// TwinCAT 3 PLC project PLC1
// ProgramVersion: 3.1.4023.0
// libraries:
//   HomePLC Alarm Manager, * (Tom Oyen)
//   HomePLC DIO, * (Tom Oyen)
//   HomePLC Home, * (Tom Oyen)
//   HomePLC Logging, * (Tom Oyen)
//   Tc2_Standard, * (Beckhoff Automation GmbH)
//   Tc2_System, * (Beckhoff Automation GmbH)
//   Tc3_Module, * (Beckhoff Automation GmbH)
//   VisuDialogs, * (System)
//   HomePLC Link Manager,newest,Tom Oyen
// project tree:
//   / Class Diagram.TcCD (not stored), GlobalTextList.TcGTLO, PlcTask.TcTTO, Visualization Manager.TcVMO (not stored)
//   DUTs/Areas/ ST_Area_DiningRoom.TcDUT, ST_Area_Bedroom2.TcDUT, ST_Area_Toilet2.TcDUT, ST_Area_Bathroom.TcDUT, ST_Area_Bedroom1.TcDUT, ST_Area_Entrance.TcDUT, ST_Area_Kitchen.TcDUT, ST_Area_StorageRoom.TcDUT, ST_Area_Toilet1.TcDUT, ST_Area_LivingRoom.TcDUT
//   DUTs/Floors/ ST_Floor_FirstFloor.TcDUT, ST_Floor_SecondFloor.TcDUT
//   DUTs/Wall plates/ ST_WP_EntranceDoor.TcDUT, ST_WP_EntranceStairs.TcDUT, ST_WP_StorageRoom.TcDUT, ST_WP_Bathroom.TcDUT, ST_WP_Bedroom1.TcDUT, ST_WP_Bedroom1BedR.TcDUT, ST_WP_Bedroom1BedL.TcDUT, ST_WP_Bedroom2.TcDUT, ST_WP_Toilet2.TcDUT, ST_WP_LivingRoom.TcDUT, ST_WP_Toilet1.TcDUT, ST_WP_DiningRoom.TcDUT, ST_WP_Kitchen.TcDUT
//   GVLs/ IO.TcGVL
//   POUs/General/Implicit checks/ CheckBounds.TcPOU, CheckDivDInt.TcPOU, CheckDivLInt.TcPOU, CheckDivLReal.TcPOU, CheckDivReal.TcPOU, CheckLRangeSigned.TcPOU, CheckLRangeUnsigned.TcPOU, CheckPointer.TcPOU, CheckRangeSigned.TcPOU, CheckRangeUnsigned.TcPOU
//   POUs/Home/ FB_MyHome.TcPOU
//   POUs/ MAIN.TcPOU
//   POUs/Simulation/ FB_ButtonSim.TcPOU, FB_Simulation.TcPOU
//   VISUs/ Alarm.TcVIS, LinkInfo.TcVIS, Overview.TcVIS
// real-time tasks:
//   TASK PlcTask: cycle T#10ms, priority 20, ADS port 350
//   TASK VISU_TASK: cycle T#200000us, priority 30, ADS port 351

CONFIGURATION PLC1
    RESOURCE PLC ON TwinCAT3
        TASK PlcTask(INTERVAL := T#10ms, PRIORITY := 20);
        PROGRAM MAIN WITH PlcTask : MAIN;
    END_RESOURCE
END_CONFIGURATION

// ---- DUTs/Areas/ST_Area_DiningRoom.TcDUT
TYPE ST_Area_DiningRoom :
STRUCT
	wpRoom				: ST_WP_DiningRoom;
	fbSpotLights		: FB_DigitalOut;
	fbCenterLight		: FB_DigitalOut;
	fbAlarmsensor		: FB_AlarmSensor(sSensorName := 'DiningRoom', bEnableWarning := TRUE);
END_STRUCT
END_TYPE

// ---- DUTs/Areas/ST_Area_Bedroom2.TcDUT
TYPE ST_Area_Bedroom2 :
STRUCT
	wpRoom				: ST_WP_Bedroom2;
	fbSpotLights		: FB_DigitalOut;
END_STRUCT
END_TYPE

// ---- DUTs/Areas/ST_Area_Toilet2.TcDUT
TYPE ST_Area_Toilet2 :
STRUCT
	wpRuimte			: ST_WP_Toilet2;		// WC2 B1L0
	fbLichtSpot			: FB_DigitalOut;	// Licht spot + nis spot
END_STRUCT
END_TYPE

// ---- DUTs/Areas/ST_Area_Bathroom.TcDUT
TYPE ST_Area_Bathroom :
STRUCT
	wpRoom				: ST_WP_Bathroom;
	fbSpotLights		: FB_DigitalOut;
	fbSinkLights		: FB_DigitalOut;
END_STRUCT
END_TYPE

// ---- DUTs/Areas/ST_Area_Bedroom1.TcDUT
TYPE ST_Area_Bedroom1 :
STRUCT
	wpRoom				: ST_WP_Bedroom1;
	wpBedL				: ST_WP_Bedroom1BedL;
	fbSocketBedL		: FB_DigitalOut;
	wpBedR				: ST_WP_Bedroom1BedR;
	fbSocketBedR		: FB_DigitalOut;
	fbSpotLights		: FB_DigitalOut;
END_STRUCT
END_TYPE

// ---- DUTs/Floors/ST_Floor_FirstFloor.TcDUT
TYPE ST_Floor_FirstFloor :
STRUCT
	Entrance			: ST_Area_Entrance;
	Toilet1				: ST_Area_Toilet1;
	LivingRoom			: ST_Area_LivingRoom;
	DiningRoom			: ST_Area_DiningRoom;
	Kitchen				: ST_Area_Kitchen;
	StorageRoom			: ST_Area_StorageRoom;
END_STRUCT
END_TYPE

// ---- DUTs/Floors/ST_Floor_SecondFloor.TcDUT
TYPE ST_Floor_SecondFloor :
STRUCT
	Toilet2				: ST_Area_Toilet2;
	Bathroom			: ST_Area_Bathroom;
	Bedroom1			: ST_Area_Bedroom1;
	Bedroom2			: ST_Area_Bedroom2;
END_STRUCT
END_TYPE

// ---- DUTs/Areas/ST_Area_Entrance.TcDUT
TYPE ST_Area_Entrance :
STRUCT
	wpDoor				: ST_WP_EntranceDoor;
	fbAlarmPanel		: FB_AlarmKeypad(sKeypadName := 'Entrance');
	wpStairs			: ST_WP_EntranceStairs;
	fbSpotLights		: FB_DigitalOut;
	fbAlarmSensor		: FB_AlarmSensor(sSensorName := 'Entrance', bEnableWarning := TRUE);
	fbAlarmSiren		: FB_AlarmSiren(sSirenName := 'Entrance');
END_STRUCT
END_TYPE

// ---- DUTs/Areas/ST_Area_Kitchen.TcDUT
TYPE ST_Area_Kitchen :
STRUCT
	wpRoom				: ST_WP_Kitchen;
	fbLightIsland		: FB_DigitalOut;
	fbCenterLight		: FB_DigitalOut;
	fbSocket			: FB_DigitalOut;
	fbAlarmSensor		: FB_AlarmSensor(sSensorName := 'Kitchen', bEnableWarning := TRUE);
END_STRUCT
END_TYPE

// ---- DUTs/Areas/ST_Area_StorageRoom.TcDUT
TYPE ST_Area_StorageRoom :
STRUCT
	wpRoom				: ST_WP_StorageRoom;
	fbSpotLights		: FB_DigitalOut;
	fbAlarmsensor		: FB_AlarmSensor(sSensorName := 'StorageRoom', bEnableWarning := FALSE);
END_STRUCT
END_TYPE

// ---- DUTs/Areas/ST_Area_Toilet1.TcDUT
TYPE ST_Area_Toilet1 :
STRUCT
	wpRoom				: ST_WP_Toilet1;
	fbSpotLight			: FB_DigitalOut;
END_STRUCT
END_TYPE

// ---- DUTs/Areas/ST_Area_LivingRoom.TcDUT
TYPE ST_Area_LivingRoom :
STRUCT
	wpRoom			: ST_WP_LivingRoom;
	fbSpotLights	: FB_DigitalOut;
	fbAlarmSensor	: FB_AlarmSensor(sSensorName := 'LivingRoom', bEnableWarning := FALSE);
END_STRUCT
END_TYPE

// ---- DUTs/Wall plates/ST_WP_EntranceDoor.TcDUT
// Inkom deur - B11-11L11-11
TYPE ST_WP_EntranceDoor :
STRUCT
	fbButton1		: FB_DigitalIn;
	fbLed1			: FB_DigitalOut;
	fbButton2		: FB_DigitalIn;
	fbLed2			: FB_DigitalOut;
	fbButton3		: FB_DigitalIn;
	fbLed3			: FB_DigitalOut;
	fbButton4		: FB_DigitalIn;
	fbLed4			: FB_DigitalOut;
END_STRUCT
END_TYPE

// ---- DUTs/Wall plates/ST_WP_EntranceStairs.TcDUT
// Inkom trap B1-11L0-00
TYPE ST_WP_EntranceStairs :
STRUCT
	fbButton1		: FB_DigitalIn;
	fbButton2		: FB_DigitalIn;
	fbButton3		: FB_DigitalIn;
END_STRUCT
END_TYPE

// ---- DUTs/Wall plates/ST_WP_StorageRoom.TcDUT
// Bergplaats B1-11L0-00
TYPE ST_WP_StorageRoom :
STRUCT
	fbButton1		: FB_DigitalIn;
	fbButton2		: FB_DigitalIn;
	fbButton3		: FB_DigitalIn;
END_STRUCT
END_TYPE

// ---- DUTs/Wall plates/ST_WP_Bathroom.TcDUT
// Badkamer meubel B1L0
TYPE ST_WP_Bathroom :
STRUCT
	fbKnop1		: FB_DigitalIn;
END_STRUCT
END_TYPE

// ---- DUTs/Wall plates/ST_WP_Bedroom1.TcDUT
// Slaapkamer 1 B1-1L0-0
TYPE ST_WP_Bedroom1 :
STRUCT
	fbButton1		: FB_DigitalIn;
	fbButton2		: FB_DigitalIn;
END_STRUCT
END_TYPE

// ---- DUTs/Wall plates/ST_WP_Bedroom1BedR.TcDUT
// Slaapkamer 1 bed R B11L00
TYPE ST_WP_Bedroom1BedR :
STRUCT
	fbButton1		: FB_DigitalIn;
	fbButton2		: FB_DigitalIn;
END_STRUCT
END_TYPE

// ---- DUTs/Wall plates/ST_WP_Bedroom1BedL.TcDUT
// Slaapkamer 1 bed L B11L00
TYPE ST_WP_Bedroom1BedL :
STRUCT
	fbButton1		: FB_DigitalIn;
	fbButton2		: FB_DigitalIn;
END_STRUCT
END_TYPE

// ---- DUTs/Wall plates/ST_WP_Bedroom2.TcDUT
// Slaapkamer 2 B1L0
TYPE ST_WP_Bedroom2 :
STRUCT
	fbButton1		: FB_DigitalIn;
END_STRUCT
END_TYPE

// ---- DUTs/Wall plates/ST_WP_Toilet2.TcDUT
// WC2 B1L0
TYPE ST_WP_Toilet2 :
STRUCT
	fbButton1		: FB_DigitalIn;
END_STRUCT
END_TYPE

// ---- DUTs/Wall plates/ST_WP_LivingRoom.TcDUT
// Zithoek B11-11L00-00
TYPE ST_WP_LivingRoom :
STRUCT
	fbButton1		: FB_DigitalIn;
	fbButton2		: FB_DigitalIn;
	fbButton3		: FB_DigitalIn;
	fbButton4		: FB_DigitalIn;
END_STRUCT
END_TYPE

// ---- DUTs/Wall plates/ST_WP_Toilet1.TcDUT
// WC1 B1L0
TYPE ST_WP_Toilet1 :
STRUCT
	fbButton1		: FB_DigitalIn;
END_STRUCT
END_TYPE

// ---- DUTs/Wall plates/ST_WP_DiningRoom.TcDUT
// Eethoek B1-1-11L0-0-00
TYPE ST_WP_DiningRoom :
STRUCT
	fbKnop1		: FB_DigitalIn;
	fbKnop2		: FB_DigitalIn;
	fbKnop3		: FB_DigitalIn;
	fbKnop4		: FB_DigitalIn;
END_STRUCT
END_TYPE

// ---- DUTs/Wall plates/ST_WP_Kitchen.TcDUT
// Keuken B1-11-11L0-00-00
TYPE ST_WP_Kitchen :
STRUCT
	fbButton1		: FB_DigitalIn;
	fbButton2		: FB_DigitalIn;
	fbButton3		: FB_DigitalIn;
	fbButton4		: FB_DigitalIn;
	fbButton5		: FB_DigitalIn;
END_STRUCT
END_TYPE

// ---- GVLs/IO.TcGVL
{attribute 'qualified_only'}
VAR_GLOBAL
	// IO
	FirstFloor		: ST_Floor_FirstFloor;
	SecondFloor		: ST_Floor_SecondFloor;
END_VAR

// ---- POUs/MAIN.TcPOU
// Home PLC
PROGRAM MAIN
VAR
	fbHome			: FB_MyHome;
	fbSimulation	: FB_Simulation;
END_VAR

fbHome.Execute();
//fbSimulation.Execute();

END_PROGRAM

// ---- POUs/Home/FB_MyHome.TcPOU
// Home implementation
FUNCTION_BLOCK FB_MyHome EXTENDS FB_Home
VAR
	// IO groups
	fbDIGroupAllOff		: FB_DIGroup;		// Input group containing all inputs for the all-off function
	fbDOGroupAllOff		: FB_DOGroup;		// Output group containing all outputs for the all-off function
END_VAR

// Configure
METHOD PROTECTED Configure
CreateDIGroupAllOff(IDIGroup := fbDIGroupAllOff);
CreateDOGroupAllOff(IDOGroup := fbDOGroupAllOff);

SUPER^.Configure();
END_METHOD

// Configure alarm
METHOD PROTECTED ConfigureAlarm
VAR_INPUT
	IAlarmManager	: I_AlarmManager;		// Alarm manager interface
END_VAR
IAlarmManager.AddKeypad(IKeyPad := IO.FirstFloor.Entrance.fbAlarmPanel);

IAlarmManager.AddSensor(ISensor := IO.FirstFloor.Entrance.fbAlarmSensor);
IAlarmManager.AddSensor(ISensor := IO.FirstFloor.LivingRoom.fbAlarmSensor);
IAlarmManager.AddSensor(ISensor := IO.FirstFloor.DiningRoom.fbAlarmsensor);
IAlarmManager.AddSensor(ISensor := IO.FirstFloor.Kitchen.fbAlarmSensor);
IAlarmManager.AddSensor(ISensor := IO.FirstFloor.StorageRoom.fbAlarmsensor);

IAlarmManager.AddSiren(ISiren := IO.FirstFloor.Entrance.fbAlarmSiren);
END_METHOD

// Add links
METHOD PROTECTED ConfigureLinks
VAR_INPUT
	ILinkManager	: I_LinkManager;		// Link manager interface
END_VAR
// All off
ILinkManager.Link.InputGroup := fbDIGroupAllOff;
ILinkManager.Link.OutputGroup := fbDOGroupAllOff;
ILinkManager.Link.OutputReaction.OnHold := E_DOCommand.Off;
ILinkManager.Link.ExcludeFromOverview := TRUE;
ILinkManager.CommitLink();

// First floor - entrance spot lights
ILinkManager.Link.InputGroup.AddInput(IO.FirstFloor.Entrance.wpDoor.fbButton4);
ILinkManager.Link.InputGroup.AddInput(IO.FirstFloor.Entrance.wpStairs.fbButton3);
ILinkManager.Link.InputGroup.AddInput(IO.FirstFloor.StorageRoom.wpRoom.fbButton1);
ILinkManager.Link.OutputReaction.OnShortPress := E_DOCommand.Toggle;
ILinkManager.Link.OutputGroup.AddOutput(IO.FirstFloor.Entrance.fbSpotLights);
ILinkManager.Link.OutputGroup.AddIndicator(IO.FirstFloor.Entrance.wpDoor.fbLed4);
ILinkManager.CommitLink();

// First floor - WC1 spot light
ILinkManager.Link.InputGroup.AddInput(IO.FirstFloor.Toilet1.wpRoom.fbButton1);
ILinkManager.Link.OutputReaction.OnShortPress := E_DOCommand.Toggle;
ILinkManager.Link.OutputGroup.AddOutput(IO.FirstFloor.Toilet1.fbSpotLight);
ILinkManager.CommitLink();

// First floor - Living room spot lights
ILinkManager.Link.InputGroup.AddInput(IO.FirstFloor.LivingRoom.wpRoom.fbButton4);
ILinkManager.Link.InputGroup.AddInput(IO.FirstFloor.DiningRoom.wpRoom.fbKnop4);
ILinkManager.Link.InputGroup.AddInput(IO.FirstFloor.Entrance.wpStairs.fbButton2);
ILinkManager.Link.OutputReaction.OnShortPress := E_DOCommand.Toggle;
ILinkManager.Link.OutputGroup.AddOutput(IO.FirstFloor.LivingRoom.fbSpotLights);
ILinkManager.CommitLink();

// First floor - Dining room spot lights
ILinkManager.Link.InputGroup.AddInput(IO.FirstFloor.DiningRoom.wpRoom.fbKnop3);
ILinkManager.Link.InputGroup.AddInput(IO.FirstFloor.LivingRoom.wpRoom.fbButton1);
ILinkManager.Link.OutputReaction.OnShortPress := E_DOCommand.Toggle;
ILinkManager.Link.OutputGroup.AddOutput(IO.FirstFloor.DiningRoom.fbSpotLights);
ILinkManager.CommitLink();

// First floor - Dining room center light
ILinkManager.Link.InputGroup.AddInput(IO.FirstFloor.DiningRoom.wpRoom.fbKnop2);
ILinkManager.Link.InputGroup.AddInput(IO.FirstFloor.LivingRoom.wpRoom.fbButton2);
ILinkManager.Link.OutputReaction.OnShortPress := E_DOCommand.Toggle;
ILinkManager.Link.OutputGroup.AddOutput(IO.FirstFloor.DiningRoom.fbCenterLight);
ILinkManager.CommitLink();

// First floor - Kitchen island lights
ILinkManager.Link.InputGroup.AddInput(IO.FirstFloor.Kitchen.wpRoom.fbButton4);
ILinkManager.Link.OutputReaction.OnShortPress := E_DOCommand.Toggle;
ILinkManager.Link.OutputGroup.AddOutput(IO.FirstFloor.Kitchen.fbLightIsland);
ILinkManager.CommitLink();

// First floor - Kitchen center light
ILinkManager.Link.InputGroup.AddInput(IO.FirstFloor.Kitchen.wpRoom.fbButton2);
ILinkManager.Link.OutputReaction.OnShortPress := E_DOCommand.Toggle;
ILinkManager.Link.OutputGroup.AddOutput(IO.FirstFloor.Kitchen.fbCenterLight);
ILinkManager.CommitLink();

// First floor - Kitchen socket
ILinkManager.Link.InputGroup.AddInput(IO.FirstFloor.Kitchen.wpRoom.fbButton5);
ILinkManager.Link.OutputReaction.OnShortPress := E_DOCommand.Toggle;
ILinkManager.Link.OutputGroup.AddOutput(IO.FirstFloor.Kitchen.fbSocket);
ILinkManager.CommitLink();

// First floor - Storage room spot lights
ILinkManager.Link.InputGroup.AddInput(IO.FirstFloor.StorageRoom.wpRoom.fbButton2);
ILinkManager.Link.OutputReaction.OnShortPress := E_DOCommand.Toggle;
ILinkManager.Link.OutputGroup.AddOutput(IO.FirstFloor.StorageRoom.fbSpotLights);
ILinkManager.CommitLink();

// Second floor - WC2 spots
ILinkManager.Link.InputGroup.AddInput(IO.SecondFloor.Toilet2.wpRuimte.fbButton1);
ILinkManager.Link.OutputReaction.OnShortPress := E_DOCommand.Toggle;
ILinkManager.Link.OutputGroup.AddOutput(IO.SecondFloor.Toilet2.fbLichtSpot);
ILinkManager.CommitLink();

// Second floor - Bathroom sink lights
ILinkManager.Link.InputGroup.AddInput(IO.SecondFloor.Bathroom.wpRoom.fbKnop1);
ILinkManager.Link.OutputReaction.OnShortPress := E_DOCommand.Toggle;
ILinkManager.Link.OutputGroup.AddOutput(IO.SecondFloor.Bathroom.fbSinkLights);
ILinkManager.CommitLink();

// Second floor - Bedroom 1 spot lights
ILinkManager.Link.InputGroup.AddInput(IO.SecondFloor.Bedroom1.wpRoom.fbButton2);
ILinkManager.Link.InputGroup.AddInput(IO.SecondFloor.Bedroom1.wpBedL.fbButton1);
ILinkManager.Link.InputGroup.AddInput(IO.SecondFloor.Bedroom1.wpBedR.fbButton2);
ILinkManager.Link.OutputReaction.OnShortPress := E_DOCommand.Toggle;
ILinkManager.Link.OutputGroup.AddOutput(IO.SecondFloor.Bedroom1.fbSpotLights);
ILinkManager.CommitLink();

// Second floor - Bedroom 1 socket L
ILinkManager.Link.InputGroup.AddInput(IO.SecondFloor.Bedroom1.wpBedL.fbButton2);
ILinkManager.Link.OutputReaction.OnShortPress := E_DOCommand.Toggle;
ILinkManager.Link.OutputGroup.AddOutput(IO.SecondFloor.Bedroom1.fbSocketBedL);
ILinkManager.CommitLink();

// Second floor - Bedroom 1 socket R
ILinkManager.Link.InputGroup.AddInput(IO.SecondFloor.Bedroom1.wpBedR.fbButton1);
ILinkManager.Link.OutputReaction.OnShortPress := E_DOCommand.Toggle;
ILinkManager.Link.OutputGroup.AddOutput(IO.SecondFloor.Bedroom1.fbSocketBedR);
ILinkManager.CommitLink();

// Second floor - Bedroom 2 spots
ILinkManager.Link.InputGroup.AddInput(IO.SecondFloor.Bedroom2.wpRoom.fbButton1);
ILinkManager.Link.OutputReaction.OnShortPress := E_DOCommand.Toggle;
ILinkManager.Link.OutputGroup.AddOutput(IO.SecondFloor.Bedroom2.fbSpotLights);
ILinkManager.CommitLink();
END_METHOD

// Create DI group of all inputs (used to call all Execute methods)
METHOD PROTECTED CreateDIGroupAll
VAR_INPUT
	IDIGroup	: I_DIGroup;		// Digital input group interface
END_VAR
// First floor
IDIGroup.AddInput(IO.FirstFloor.StorageRoom.wpRoom.fbButton1);
IDIGroup.AddInput(IO.FirstFloor.StorageRoom.wpRoom.fbButton2);
IDIGroup.AddInput(IO.FirstFloor.StorageRoom.wpRoom.fbButton3);
IDIGroup.AddInput(IO.FirstFloor.DiningRoom.wpRoom.fbKnop1);
IDIGroup.AddInput(IO.FirstFloor.DiningRoom.wpRoom.fbKnop2);
IDIGroup.AddInput(IO.FirstFloor.DiningRoom.wpRoom.fbKnop3);
IDIGroup.AddInput(IO.FirstFloor.DiningRoom.wpRoom.fbKnop4);
IDIGroup.AddInput(IO.FirstFloor.Entrance.wpDoor.fbButton1);
IDIGroup.AddInput(IO.FirstFloor.Entrance.wpDoor.fbButton2);
IDIGroup.AddInput(IO.FirstFloor.Entrance.wpDoor.fbButton3);
IDIGroup.AddInput(IO.FirstFloor.Entrance.wpDoor.fbButton4);
IDIGroup.AddInput(IO.FirstFloor.Entrance.wpStairs.fbButton1);
IDIGroup.AddInput(IO.FirstFloor.Entrance.wpStairs.fbButton2);
IDIGroup.AddInput(IO.FirstFloor.Entrance.wpStairs.fbButton3);
IDIGroup.AddInput(IO.FirstFloor.Kitchen.wpRoom.fbButton1);
IDIGroup.AddInput(IO.FirstFloor.Kitchen.wpRoom.fbButton2);
IDIGroup.AddInput(IO.FirstFloor.Kitchen.wpRoom.fbButton3);
IDIGroup.AddInput(IO.FirstFloor.Kitchen.wpRoom.fbButton4);
IDIGroup.AddInput(IO.FirstFloor.Kitchen.wpRoom.fbButton5);
IDIGroup.AddInput(IO.FirstFloor.Toilet1.wpRoom.fbButton1);
IDIGroup.AddInput(IO.FirstFloor.LivingRoom.wpRoom.fbButton1);
IDIGroup.AddInput(IO.FirstFloor.LivingRoom.wpRoom.fbButton2);
IDIGroup.AddInput(IO.FirstFloor.LivingRoom.wpRoom.fbButton3);
IDIGroup.AddInput(IO.FirstFloor.LivingRoom.wpRoom.fbButton4);

// Verdieping
IDIGroup.AddInput(IO.SecondFloor.Bathroom.wpRoom.fbKnop1);
IDIGroup.AddInput(IO.SecondFloor.Bedroom1.wpBedL.fbButton1);
IDIGroup.AddInput(IO.SecondFloor.Bedroom1.wpBedL.fbButton2);
IDIGroup.AddInput(IO.SecondFloor.Bedroom1.wpBedR.fbButton1);
IDIGroup.AddInput(IO.SecondFloor.Bedroom1.wpBedR.fbButton2);
IDIGroup.AddInput(IO.SecondFloor.Bedroom1.wpRoom.fbButton1);
IDIGroup.AddInput(IO.SecondFloor.Bedroom1.wpRoom.fbButton2);
IDIGroup.AddInput(IO.SecondFloor.Bedroom2.wpRoom.fbButton1);
IDIGroup.AddInput(IO.SecondFloor.Toilet2.wpRuimte.fbButton1);


// Alarm
// Included here so these buttons can be used for general commands as well (e.g. all off)
IDIGroup.AddInput(IO.FirstFloor.Entrance.fbAlarmPanel.fbButton1);
IDIGroup.AddInput(IO.FirstFloor.Entrance.fbAlarmPanel.fbButton2);
IDIGroup.AddInput(IO.FirstFloor.Entrance.fbAlarmPanel.fbButton3);
IDIGroup.AddInput(IO.FirstFloor.Entrance.fbAlarmPanel.fbButton4);
IDIGroup.AddInput(IO.FirstFloor.Entrance.fbAlarmPanel.fbButton5);
IDIGroup.AddInput(IO.FirstFloor.Entrance.fbAlarmPanel.fbButton6);
END_METHOD

// Create DI group of all inputs that are used to turn all outputs off
METHOD PRIVATE CreateDIGroupAllOff
VAR_INPUT
	IDIGroup	: I_DIGroup;		// Digital input group interface
END_VAR
// Gelijkvloers
IDIGroup.AddInput(IO.FirstFloor.StorageRoom.wpRoom.fbButton1);
IDIGroup.AddInput(IO.FirstFloor.StorageRoom.wpRoom.fbButton2);
IDIGroup.AddInput(IO.FirstFloor.StorageRoom.wpRoom.fbButton3);
IDIGroup.AddInput(IO.FirstFloor.DiningRoom.wpRoom.fbKnop1);
IDIGroup.AddInput(IO.FirstFloor.DiningRoom.wpRoom.fbKnop2);
IDIGroup.AddInput(IO.FirstFloor.DiningRoom.wpRoom.fbKnop3);
IDIGroup.AddInput(IO.FirstFloor.DiningRoom.wpRoom.fbKnop4);
IDIGroup.AddInput(IO.FirstFloor.Entrance.wpDoor.fbButton1);
IDIGroup.AddInput(IO.FirstFloor.Entrance.wpDoor.fbButton2);
IDIGroup.AddInput(IO.FirstFloor.Entrance.wpDoor.fbButton3);
IDIGroup.AddInput(IO.FirstFloor.Entrance.wpDoor.fbButton4);
IDIGroup.AddInput(IO.FirstFloor.Entrance.wpStairs.fbButton1);
IDIGroup.AddInput(IO.FirstFloor.Entrance.wpStairs.fbButton2);
IDIGroup.AddInput(IO.FirstFloor.Entrance.wpStairs.fbButton3);
IDIGroup.AddInput(IO.FirstFloor.Kitchen.wpRoom.fbButton1);
IDIGroup.AddInput(IO.FirstFloor.Kitchen.wpRoom.fbButton2);
IDIGroup.AddInput(IO.FirstFloor.Kitchen.wpRoom.fbButton3);
IDIGroup.AddInput(IO.FirstFloor.Kitchen.wpRoom.fbButton4);
IDIGroup.AddInput(IO.FirstFloor.Kitchen.wpRoom.fbButton5);
IDIGroup.AddInput(IO.FirstFloor.Toilet1.wpRoom.fbButton1);
IDIGroup.AddInput(IO.FirstFloor.LivingRoom.wpRoom.fbButton1);
IDIGroup.AddInput(IO.FirstFloor.LivingRoom.wpRoom.fbButton2);
IDIGroup.AddInput(IO.FirstFloor.LivingRoom.wpRoom.fbButton3);
IDIGroup.AddInput(IO.FirstFloor.LivingRoom.wpRoom.fbButton4);

// Verdieping
IDIGroup.AddInput(IO.SecondFloor.Bathroom.wpRoom.fbKnop1);
IDIGroup.AddInput(IO.SecondFloor.Bedroom1.wpBedL.fbButton1);
IDIGroup.AddInput(IO.SecondFloor.Bedroom1.wpBedL.fbButton2);
IDIGroup.AddInput(IO.SecondFloor.Bedroom1.wpBedR.fbButton1);
IDIGroup.AddInput(IO.SecondFloor.Bedroom1.wpBedR.fbButton2);
IDIGroup.AddInput(IO.SecondFloor.Bedroom1.wpRoom.fbButton1);
IDIGroup.AddInput(IO.SecondFloor.Bedroom1.wpRoom.fbButton2);
IDIGroup.AddInput(IO.SecondFloor.Bedroom2.wpRoom.fbButton1);
IDIGroup.AddInput(IO.SecondFloor.Toilet2.wpRuimte.fbButton1);

// Alarm
IDIGroup.AddInput(IO.FirstFloor.Entrance.fbAlarmPanel.fbButton1);
IDIGroup.AddInput(IO.FirstFloor.Entrance.fbAlarmPanel.fbButton2);
IDIGroup.AddInput(IO.FirstFloor.Entrance.fbAlarmPanel.fbButton3);
IDIGroup.AddInput(IO.FirstFloor.Entrance.fbAlarmPanel.fbButton4);
IDIGroup.AddInput(IO.FirstFloor.Entrance.fbAlarmPanel.fbButton5);
IDIGroup.AddInput(IO.FirstFloor.Entrance.fbAlarmPanel.fbButton6);
END_METHOD

// Create DO group of all outputs (used to call all Execute methods)
METHOD PROTECTED CreateDOGroupAll
VAR_INPUT
	IDOGroup	: I_DOGroup;		// Digital output group interface
END_VAR
// First floor
IDOGroup.AddOutput(IO.FirstFloor.StorageRoom.fbSpotLights);
IDOGroup.AddOutput(IO.FirstFloor.DiningRoom.fbSpotLights);
IDOGroup.AddOutput(IO.FirstFloor.DiningRoom.fbCenterLight);
IDOGroup.AddOutput(IO.FirstFloor.Entrance.fbSpotLights);
IDOGroup.AddOutput(IO.FirstFloor.Entrance.wpDoor.fbLed1);
IDOGroup.AddOutput(IO.FirstFloor.Entrance.wpDoor.fbLed2);
IDOGroup.AddOutput(IO.FirstFloor.Entrance.wpDoor.fbLed3);
IDOGroup.AddOutput(IO.FirstFloor.Entrance.wpDoor.fbLed4);
IDOGroup.AddOutput(IO.FirstFloor.Kitchen.fbLightIsland);
IDOGroup.AddOutput(IO.FirstFloor.Kitchen.fbCenterLight);
IDOGroup.AddOutput(IO.FirstFloor.Kitchen.fbSocket);
IDOGroup.AddOutput(IO.FirstFloor.Toilet1.fbSpotLight);
IDOGroup.AddOutput(IO.FirstFloor.LivingRoom.fbSpotLights);

// Second floor
IDOGroup.AddOutput(IO.SecondFloor.Bathroom.fbSpotLights);
IDOGroup.AddOutput(IO.SecondFloor.Bathroom.fbSinkLights);
IDOGroup.AddOutput(IO.SecondFloor.Bedroom1.fbSpotLights);
IDOGroup.AddOutput(IO.SecondFloor.Bedroom1.fbSocketBedL);
IDOGroup.AddOutput(IO.SecondFloor.Bedroom1.fbSocketBedR);
IDOGroup.AddOutput(IO.SecondFloor.Bedroom2.fbSpotLights);
IDOGroup.AddOutput(IO.SecondFloor.Toilet2.fbLichtSpot);


// Alarm
IDOGroup.AddOutput(IO.FirstFloor.Entrance.fbAlarmPanel.fbLed1);
IDOGroup.AddOutput(IO.FirstFloor.Entrance.fbAlarmPanel.fbLed2);
IDOGroup.AddOutput(IO.FirstFloor.Entrance.fbAlarmPanel.fbLed3);
IDOGroup.AddOutput(IO.FirstFloor.Entrance.fbAlarmPanel.fbLed4);
IDOGroup.AddOutput(IO.FirstFloor.Entrance.fbAlarmPanel.fbLed5);
IDOGroup.AddOutput(IO.FirstFloor.Entrance.fbAlarmPanel.fbLed6);
IDOGroup.AddOutput(IO.FirstFloor.Entrance.fbAlarmPanel.fbBuzzer);
IDOGroup.AddOutput(IO.FirstFloor.Entrance.fbAlarmSiren.fbSiren);
IDOGroup.AddOutput(IO.FirstFloor.Entrance.fbAlarmSiren.fbLight);
END_METHOD

// Create DO group of all outputs that are turned off when all needs to be turned off
METHOD PRIVATE CreateDOGroupAllOff
VAR_INPUT
	IDOGroup	: I_DOGroup;		// Digital output group interface
END_VAR
// First floor
IDOGroup.AddOutput(IO.FirstFloor.StorageRoom.fbSpotLights);
IDOGroup.AddOutput(IO.FirstFloor.DiningRoom.fbSpotLights);
IDOGroup.AddOutput(IO.FirstFloor.DiningRoom.fbCenterLight);
IDOGroup.AddOutput(IO.FirstFloor.Entrance.fbSpotLights);
IDOGroup.AddOutput(IO.FirstFloor.Entrance.wpDoor.fbLed1);
IDOGroup.AddOutput(IO.FirstFloor.Entrance.wpDoor.fbLed2);
IDOGroup.AddOutput(IO.FirstFloor.Entrance.wpDoor.fbLed3);
IDOGroup.AddOutput(IO.FirstFloor.Entrance.wpDoor.fbLed4);
IDOGroup.AddOutput(IO.FirstFloor.Kitchen.fbLightIsland);
IDOGroup.AddOutput(IO.FirstFloor.Kitchen.fbCenterLight);
IDOGroup.AddOutput(IO.FirstFloor.Kitchen.fbSocket);
IDOGroup.AddOutput(IO.FirstFloor.Toilet1.fbSpotLight);
IDOGroup.AddOutput(IO.FirstFloor.LivingRoom.fbSpotLights);

// Verdieping
IDOGroup.AddOutput(IO.SecondFloor.Bathroom.fbSpotLights);
IDOGroup.AddOutput(IO.SecondFloor.Bathroom.fbSinkLights);
IDOGroup.AddOutput(IO.SecondFloor.Bedroom1.fbSpotLights);
IDOGroup.AddOutput(IO.SecondFloor.Bedroom1.fbSocketBedL);
IDOGroup.AddOutput(IO.SecondFloor.Bedroom1.fbSocketBedR);
IDOGroup.AddOutput(IO.SecondFloor.Bedroom2.fbSpotLights);
IDOGroup.AddOutput(IO.SecondFloor.Toilet2.fbLichtSpot);

// Alarm
IDOGroup.AddOutput(IO.FirstFloor.Entrance.fbAlarmPanel.fbBuzzer);
END_METHOD

END_FUNCTION_BLOCK

// ---- POUs/Simulation/FB_Simulation.TcPOU
FUNCTION_BLOCK FB_Simulation

METHOD Execute : BOOL
VAR_INST
	fbButton1		: FB_ButtonSim;
	fbButton2		: FB_ButtonSim;

	bShortPress1	: BOOL;
	bLongPress1		: BOOL;
	bHold1			: BOOL;
	
	bShortPress2	: BOOL;
	bLongPress2		: BOOL;
	bHold2			: BOOL;
END_VAR
fbButton1(IButton := IO.FirstFloor.Kitchen.wpRoom.fbButton1, bShortPress := bShortPress1, bLongPress := bLongPress1, bHold := bHold1);
fbButton2(IButton := IO.FirstFloor.Kitchen.wpRoom.fbButton2, bShortPress := bShortPress2, bLongPress := bLongPress2, bHold := bHold2);
END_METHOD

END_FUNCTION_BLOCK

// ---- POUs/Simulation/FB_ButtonSim.TcPOU
FUNCTION_BLOCK FB_ButtonSim
VAR_INPUT
	IButton			: I_DigitalIn;
END_VAR
VAR_IN_OUT
	bShortPress		: BOOL;
	bLongPress		: BOOL;
	bHold			: BOOL;
END_VAR
VAR
	bOut			: BOOL;
	fbTimer			: TON;
END_VAR

IF bShortPress	THEN fbTimer.PT := T#100MS; END_IF
IF bLongPress	THEN fbTimer.PT := T#500MS; END_IF
IF bHold		THEN fbTimer.PT := T#3000MS; END_IF
IF bShortPress OR bLongPress OR bHold THEN
	bOut := TRUE;
	bShortPress := FALSE;
	bLongPress := FALSE;
	bHold := FALSE;
END_IF

fbTimer(IN := bOut);
if fbTimer.Q then
	bOut := FALSE;
END_IF

IButton.SetExternalIn(bIn := bOut);

END_FUNCTION_BLOCK

// ---- POUs/General/Implicit checks/CheckBounds.TcPOU
// Implicitly generated code : DO NOT EDIT
FUNCTION CheckBounds : DINT
VAR_INPUT
	index, lower, upper: DINT;
END_VAR
// User defined local variables
VAR
    sMessageLow   : STRING := 'CheckBounds: Index too low (%d)';
    sMessageHigh  : STRING := 'CheckBounds: Index too high (%d)';
END_VAR

// This function is called every time an array is indexed
// See https://infosys.beckhoff.com/english.php?content=../content/1033/tc3_plc_intro/2530356875.html&id=

{noflow}
// Index too low
IF index < lower THEN
    CheckBounds := lower;
    // Log message
    ADSLOGDINT(msgCtrlMask := ADSLOG_MSGTYPE_WARN,
               msgFmtStr   := sMessageLow,
               dintArg     := index);

// Index too high
ELSIF index > upper THEN
    CheckBounds := upper;
    // Log message
    ADSLOGDINT(msgCtrlMask := ADSLOG_MSGTYPE_WARN,
               msgFmtStr   := sMessageHigh,
               dintArg     := index);

// Index OK
ELSE 
    CheckBounds := index;
END_IF
{flow}

END_FUNCTION

// ---- POUs/General/Implicit checks/CheckDivDInt.TcPOU
// Implicitly generated code : DO NOT EDIT
FUNCTION CheckDivDInt : DINT
VAR_INPUT
	divisor:DINT;
END_VAR
VAR
    sMessage   : STRING := 'CheckDivDInt: Division by zero (%d)';
END_VAR

// Implicitly generated code : Only an Implementation suggestion
{noflow}
IF divisor = 0 THEN
	CheckDivDInt:=1;
	// Log message
    ADSLOGDINT(msgCtrlMask := ADSLOG_MSGTYPE_WARN,
               msgFmtStr   := sMessage,
               dintArg     := divisor);
ELSE
	CheckDivDInt:=divisor;
END_IF;
{flow}

END_FUNCTION

// ---- POUs/General/Implicit checks/CheckDivLInt.TcPOU
// Implicitly generated code : DO NOT EDIT
FUNCTION CheckDivLInt : LINT
VAR_INPUT
	divisor:LINT;
END_VAR
VAR
    sMessage   : STRING := 'CheckDivLInt: Division by zero (%d)';
END_VAR

// Implicitly generated code : Only an Implementation suggestion
{noflow}
IF divisor = 0 THEN
	CheckDivLInt:=1;
	// Log message
    ADSLOGDINT(msgCtrlMask := ADSLOG_MSGTYPE_WARN,
               msgFmtStr   := sMessage,
               dintArg     := 0);
ELSE
	CheckDivLInt:=divisor;
END_IF;
{flow}

END_FUNCTION

// ---- POUs/General/Implicit checks/CheckDivLReal.TcPOU
// Implicitly generated code : DO NOT EDIT
FUNCTION CheckDivLReal : LREAL
VAR_INPUT
	divisor:LREAL;
END_VAR
VAR
    sMessage   : STRING := 'CheckDivLReal: Division by zero (%d)';
END_VAR

// Implicitly generated code : Only an Implementation suggestion
{noflow}
IF divisor = 0 THEN
	CheckDivLReal:=1;
	// Log message
    ADSLOGDINT(msgCtrlMask := ADSLOG_MSGTYPE_WARN,
               msgFmtStr   := sMessage,
               dintArg     := 0);
ELSE
	CheckDivLReal:=divisor;
END_IF;
{flow}

END_FUNCTION

// ---- POUs/General/Implicit checks/CheckDivReal.TcPOU
// Implicitly generated code : DO NOT EDIT
FUNCTION CheckDivReal : REAL
VAR_INPUT
	divisor:REAL;
END_VAR
VAR
    sMessage   : STRING := 'CheckDivReal: Division by zero (%d)';
END_VAR

// Implicitly generated code : Only an Implementation suggestion
{noflow}
IF divisor = 0 THEN
	CheckDivReal:=1;
	// Log message
    ADSLOGDINT(msgCtrlMask := ADSLOG_MSGTYPE_WARN,
               msgFmtStr   := sMessage,
               dintArg     := 0);
ELSE
	CheckDivReal:=divisor;
END_IF;
{flow}

END_FUNCTION

// ---- POUs/General/Implicit checks/CheckLRangeSigned.TcPOU
// Implicitly generated code : DO NOT EDIT
FUNCTION CheckLRangeSigned : LINT
VAR_INPUT
	value, lower, upper: LINT;
END_VAR
VAR
    sMessageLow   : STRING := 'CheckLRangeSigned: Value too low (%d)';
    sMessageHigh  : STRING := 'CheckLRangeSigned: Value too high (%d)';
END_VAR

// Implicitly generated code : Only an Implementation suggestion
{noflow}
IF (value < lower) THEN
	CheckLRangeSigned := lower;
	// Log message
    ADSLOGLREAL(msgCtrlMask := ADSLOG_MSGTYPE_WARN,
               msgFmtStr   := sMessageLow,
               lrealArg     := TO_REAL(value));
ELSIF(value > upper) THEN
	CheckLRangeSigned := upper;
	// Log message
    ADSLOGLREAL(msgCtrlMask := ADSLOG_MSGTYPE_WARN,
               msgFmtStr   := sMessageHigh,
               lrealArg     := TO_REAL(value));
ELSE
	CheckLRangeSigned := value;
END_IF

{flow}

END_FUNCTION

// ---- POUs/General/Implicit checks/CheckLRangeUnsigned.TcPOU
// Implicitly generated code : DO NOT EDIT
FUNCTION CheckLRangeUnsigned : ULINT
VAR_INPUT
	value, lower, upper: ULINT;
END_VAR
VAR
    sMessageLow   : STRING := 'CheckLRangeUnsigned: Value too low (%d)';
    sMessageHigh  : STRING := 'CheckLRangeUnsigned: Value too high (%d)';
END_VAR

// Implicitly generated code : Only an Implementation suggestion
{noflow}
IF (value < lower) THEN
	CheckLRangeUnsigned := lower;
	// Log message
    ADSLOGLREAL(msgCtrlMask := ADSLOG_MSGTYPE_WARN,
               msgFmtStr   := sMessageLow,
               lrealArg     := TO_REAL(value));
ELSIF(value > upper) THEN
	CheckLRangeUnsigned := upper;
	// Log message
    ADSLOGLREAL(msgCtrlMask := ADSLOG_MSGTYPE_WARN,
               msgFmtStr   := sMessageHigh,
               lrealArg     := TO_REAL(value));
ELSE
	CheckLRangeUnsigned := value;
END_IF
{flow}

END_FUNCTION

// ---- POUs/General/Implicit checks/CheckPointer.TcPOU
// Implicitly generated code : DO NOT EDIT
FUNCTION CheckPointer : POINTER TO BYTE
VAR_INPUT 
	ptToTest : POINTER TO BYTE; // Destination address of the pointer
	iSize : DINT;		        // Size of the type the pointer points to. (e.g: 20 for POINTER TO ARRAY [0..9] OF INT) 
	iGran : DINT;		        // Granularity of the pointer access. This is the size of the biggest non-structured data type in the type the pointer points to. (e.g: 2 for POINTER TO ARRAY [0..9] OF INT)
	bWrite: BOOL;		        // Indicates read or write Access. TRUE = write access.
END_VAR

// Implicitly generated code : Only an Implementation suggestion
{noflow}
IF ptToTest=0 THEN
    ADSLOGSTR(ADSLOG_MSGTYPE_ERROR OR ADSLOG_MSGTYPE_STRING,'CheckPointer failed due to invalid address.','');
ELSIF iSize<=0 THEN
    ADSLOGSTR(ADSLOG_MSGTYPE_ERROR OR ADSLOG_MSGTYPE_STRING,'CheckPointer failed due to invalid size.','');
ELSIF iGran<=0 THEN
    ADSLOGSTR(ADSLOG_MSGTYPE_ERROR OR ADSLOG_MSGTYPE_STRING,'CheckPointer failed due to invalid granularity.','');
// -> Please note that the following memory area check is time consuming:
//ELSIF F_CheckMemoryArea(pData:=ptToTest,nSize:=DINT_TO_UDINT(iSize)) = E_TcMemoryArea.Unknown THEN
//    ADSLOGSTR(ADSLOG_MSGTYPE_ERROR OR ADSLOG_MSGTYPE_STRING,'CheckPointer failed due to unknown memory area.','');
END_IF
CheckPointer := ptToTest;
{flow}

END_FUNCTION

// ---- POUs/General/Implicit checks/CheckRangeSigned.TcPOU
// Implicitly generated code : DO NOT EDIT
FUNCTION CheckRangeSigned : DINT
VAR_INPUT
	value, lower, upper: DINT;
END_VAR
VAR
    sMessageLow   : STRING := 'CheckRangeSigned: Value too low (%d)';
    sMessageHigh  : STRING := 'CheckRangeSigned: Value too high (%d)';
END_VAR

// Implicitly generated code : Only an Implementation suggestion
{noflow}
IF (value < lower) THEN
	CheckRangeSigned := lower;
    // Log message
    ADSLOGDINT(msgCtrlMask := ADSLOG_MSGTYPE_WARN,
               msgFmtStr   := sMessageLow,
               dintArg     := value);
ELSIF(value > upper) THEN
	CheckRangeSigned := upper;
	// Log message
    ADSLOGDINT(msgCtrlMask := ADSLOG_MSGTYPE_WARN,
               msgFmtStr   := sMessageHigh,
               dintArg     := value);
ELSE
	CheckRangeSigned := value;
END_IF
{flow}

END_FUNCTION

// ---- POUs/General/Implicit checks/CheckRangeUnsigned.TcPOU
// Implicitly generated code : DO NOT EDIT
FUNCTION CheckRangeUnsigned : UDINT
VAR_INPUT
	value, lower, upper: UDINT;
END_VAR
VAR
    sMessageLow   : STRING := 'CheckRangeUnsigned: Value too low (%d)';
    sMessageHigh  : STRING := 'CheckRangeUnsigned: Value too high (%d)';
END_VAR

// Implicitly generated code : Only an Implementation suggestion
{noflow}
IF (value < lower) THEN
	CheckRangeUnsigned := lower;
	// Log message
	ADSLOGDINT(msgCtrlMask := ADSLOG_MSGTYPE_WARN,
               msgFmtStr   := sMessageLow,
               dintArg     := TO_INT(value));
ELSIF(value > upper) THEN
	CheckRangeUnsigned := upper;
	// Log message
    ADSLOGDINT(msgCtrlMask := ADSLOG_MSGTYPE_WARN,
               msgFmtStr   := sMessageHigh,
               dintArg     := TO_INT(value));
ELSE
	CheckRangeUnsigned := value;
END_IF
{flow}

END_FUNCTION

// ---- GlobalTextList.TcGTLO
TEXTLIST GlobalTextList
  976 = '%d inputs'
  584 = '%d links'
  87 = '%d outputs'
  426 = '%s'
  273 = '%s links'
  221 = '1'
  170 = '2'
  836 = '3'
  541 = '4'
  607 = '5'
  496 = '6'
  701 = 'a'
  859 = 'abcdefghij'
  280 = 'abcdefghijabcdefghijabcdefghijabcdefghijabcdefghijabcdefghijabcdefghijabcdefghijabcdefghijabcdefghabcdefghijabcdefghijabcdefghijabcdefghijabcdefghijabcdefghijabcdefghijabcdefghijabcdefghijabcdefghijabcdefghijabcdefghijabcdefghijabcdefghijabcdefghijabcdefghijabcdefghijabcdefghijabcdefghijabcdefghijabcdefghijabcdefghijabcdefghijabcdefghijabcdefghijabcdefghijabcdefghijabcdefghijabcdefghijabcdefghijijabcdefghijabcdefghijabcdefghijabcdefghijabcdefghijabcdefghijabcdefghijabcdefghijabcdefghijabcdefghijabcdefghijabcdefghijabcdefghijabcdefghijabcdefghijabcdefghijabcdefghijabcdefghijabcdefghijabcdefghijabcdefghijabcdefghijabcdefghijabcdefghijabcdefghijabcdefghijabcdefghijabcdefghijabcdefghijabcdefghijabcdefghijabcdefghijabcdefghijabcdefghijabcdefghijabcdefghijabcdefghijabcdefghijabcdefghijabcdefghijabcdefghijabcdefghijabcdefghijabcdefghijabcdefghijabcdefghijabcdefghijabcdefghijabcdefghijabcdefghijabcdefghijabcdefghijabcdefghijabcdefghijabcdefghijabcdefghijabcdefghijabcdefghijabcdefghijabcdefghijabcdefghijabcdefghijabcdefghijabcdefghijabcdefghijabcdefghijabcdefghijabcdefghijabcdefghijabcdefghijabcdefghijabcdefghijabcdefghijabcdefghijabcdefghijabcdefghijabcdefghijabcdefghijabcdefghijabcdefghijabcdefghijabcdefghijabcdefghijabcdefghijabcdefghij'
  247 = 'abcdefghijabcdefghijabcdefghijabcdefghijabcdefghijabcdefghijabcdefghijabcdefghijabcdefghijabcdefghijabcdefghijabcdefghijabcdefghijabcdefghijabcdefghijabcdefghijabcdefghijabcdefghijabcdefghijabcdefghijabcdefghijabcdefghijabcdefghijabcdefghijabcdefghijabcdefghij'
  312 = 'abcdefghijabcdefghijabcdefghijabcdefghijabcdefghijabcdefghijabcdefghijabcdefghijabcdefghijabcdefghijabcdefghijabcdefghijabcdefghijabcdefghijabcdefghijabcdefghijabcdefghijabcdefghijabcdefghijabcdefghijabcdefghijabcdefghijabcdefghijabcdefghijabcdefghijabcdefghijabcdefghijabcdefghijabcdefghijabcdefghijabcdefghijabcdefghijabcdefghijabcdefghijabcdefghijabcdefghijabcdefghijabcdefghijabcdefghijabcdefghijabcdefghijabcdefghijabcdefghijabcdefghijabcdefghijabcdefghijabcdefghijabcdefghijabcdefghijabcdefghijabcdefghijabcdefghijabcdefghijabcdefghijabcdefghijabcdefghijabcdefghijabcdefghijabcdefghijabcdefghijabcdefghijabcdefghijabcdefghijabcdefghijabcdefghijabcdefghijabcdefghijabcdefghijabcdefghijabcdefghijabcdefghijabcdefghijabcdefghijabcdefghijabcdefghijabcdefghijabcdefghabcdefghijabcdefghijabcdefghijabcdefghijabcdefghijabcdefghijabcdefghijabcdefghijabcdefghijabcdefghijabcdefghijabcdefghijabcdefghijabcdefghijabcdefghijabcdefghijabcdefghijabcdefghijabcdefghijabcdefghijabcdefghijabcdefghijabcdefghijabcdefghijabcdefghijabcdefghijabcdefghijabcdefghijabcdefghijabcdefghijijabcdefghijabcdefghijabcdefghijabcdefghijabcdefghijabcdefghijabcdefghijabcdefghijabcdefghijabcdefghijabcdefghijabcdefghijabcdefghijabcdefghijabcdefghijabcdefghijabcdefghijabcdefghijabcdefghijabcdefghijabcdefghijabcdefghijabcdefghijabcdefghijabcdefghijabcdefghijabcdefghijabcdefghijabcdefghijabcdefghijabcdefghijabcdefghijabcdefghijabcdefghijabcdefghijabcdefghijabcdefghijabcdefghijabcdefghijabcdefghijabcdefghijabcdefghijabcdefghijabcdefghijabcdefghijabcdefghijabcdefghijabcdefghijabcdefghijabcdefghijabcdefghijabcdefghijabcdefghijabcdefghijabcdefghijabcdefghijabcdefghijabcdefghijabcdefghijabcdefghijabcdefghijabcdefghijabcdefghijabcdefghijabcdefghijabcdefghijabcdefghijabcdefghijabcdefghijabcdefghijabcdefghijabcdefghijabcdefghijabcdefghijabcdefghijabcdefghijabcdefghijabcdefghijabcdefghijabcdefghijabcdefghijabcdefghijabcdefghijabcdefghijabcdefghij'
  946 = 'abcdefghijabcdefghijabcdefghijabcdefghijabcdefghijabcdefghijabcdefghijabcdefghijabcdefghijabcdefghijabcdefghijabcdefghijabcdefghijabcdefghijabcdefghijabcdefghijabcdefghijabcdefghijabcdefghijabcdefghijabcdefghijabcdefghijabcdefghijabcdefghijabcdefghijabcdefghijabcdefghijabcdefghijabcdefghijabcdefghijabcdefghijabcdefghijabcdefghijabcdefghijabcdefghijabcdefghijabcdefghijabcdefghijabcdefghijabcdefghijabcdefghijabcdefghijabcdefghijabcdefghijabcdefghijabcdefghijabcdefghijabcdefghijabcdefghijabcdefghijabcdefghijabcdefghijabcdefghijabcdefghijabcdefghijabcdefghijabcdefghijabcdefghijabcdefghijabcdefghijabcdefghijabcdefghijabcdefghijabcdefghijabcdefghijabcdefghijabcdefghijabcdefghijabcdefghijabcdefghijabcdefghijabcdefghijabcdefghijabcdefghijabcdefghijabcdefghijabcdefghijabcdefghijabcdefghijabcdefghijabcdefghijabcdefghijabcdefghijabcdefghijabcdefghijabcdefghijabcdefghijabcdefghijabcdefghijabcdefghijabcdefghijabcdefghijabcdefghijabcdefghijabcdefghij'
  981 = 'Alarm'
  332 = 'Button'
  950 = 'Buzzer'
  188 = 'Check if every input is used at least once'
  33 = 'Check if every input is used for only one output (excluding its own LED)'
  986 = 'Check if every output is controlled by one or more inputs'
  945 = 'Checkbox'
  21 = 'Enabled'
  969 = 'Inputs'
  547 = 'Light'
  234 = 'Linked inputs'
  187 = 'Linked outputs'
  734 = 'Name'
  488 = 'Only active'
  746 = 'Output'
  389 = 'Outputs'
  717 = 'Sensor'
  895 = 'Sensor alarm'
  302 = 'Sensor tamper'
  213 = 'Siren'
  204 = 'Siren tamper'
  259 = 'State'
  624 = 'Tamper'
  473 = 'Value'
END_TEXTLIST

// ---- VISUs/Alarm.TcVIS
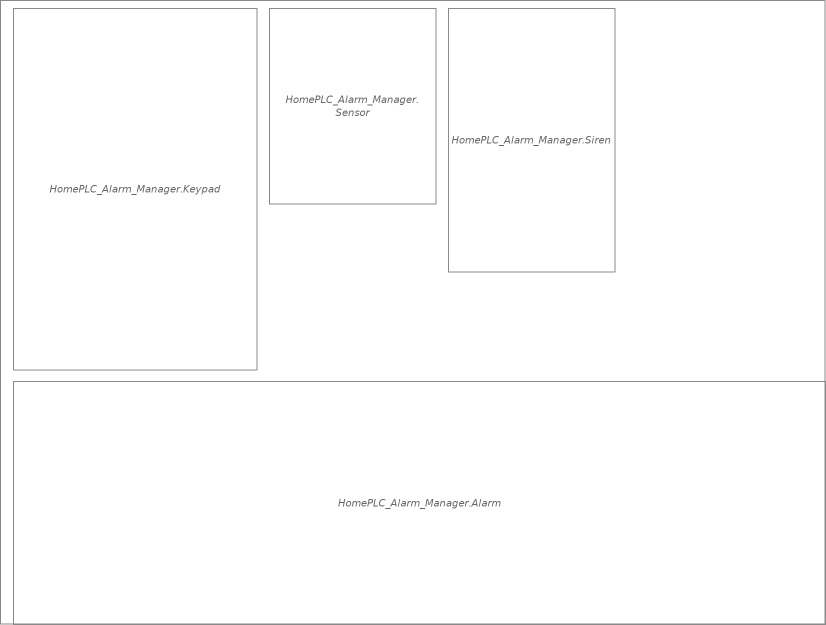
VISUALIZATION Alarm  // 826x625
    Frame (13,8 244x362)
        shows HomePLC_Alarm_Manager.Keypad(stKeypadVirtual := IO.FirstFloor.Entrance.fbAlarmPanel.stVirtual, stKeypad := IO.FirstFloor.Entrance.fbAlarmPanel.stHMI)
    Frame (13,381 813x244)
        shows HomePLC_Alarm_Manager.Alarm(stAlarm := MAIN.fbHome.fbAlarmManager.stHMI)
    Frame (269,8 167x196)
        shows HomePLC_Alarm_Manager.Sensor(stSensor := IO.FirstFloor.Entrance.fbAlarmSensor.stHMI)
    Frame (448,8 167x264)
        shows HomePLC_Alarm_Manager.Siren(stSiren := IO.FirstFloor.Entrance.fbAlarmSiren.stHMI)
END_VISUALIZATION

// ---- VISUs/LinkInfo.TcVIS
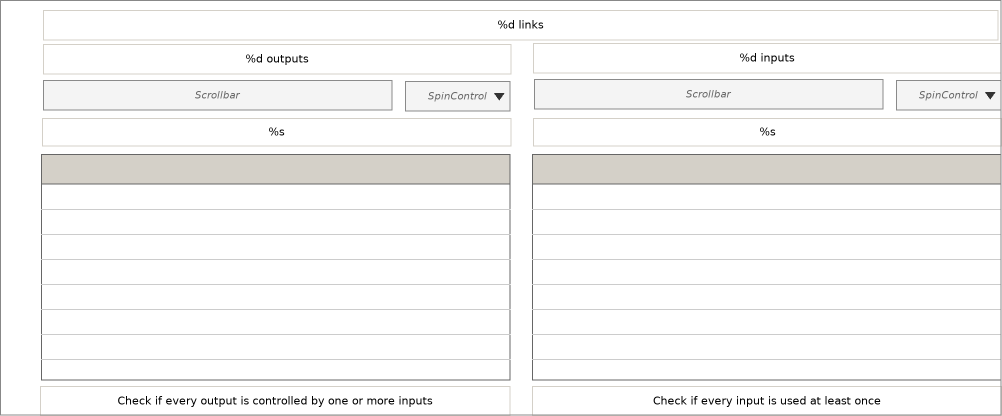
VISUALIZATION LinkInfo  // 1002x416
    Table (41,154 469x226), data array: MAIN.fbHome.stHmi.aLinkedInputs
        p3854506369: MAIN.fbHome.stHmi.aLinkedInputs[INDEX]
        p2232123230: Linked inputs
    Textfield (42,118 469x28), "%s", text variable: MAIN.fbHome.stHmi.sOutput
    SpinControl (405,81 105x30), variable: MAIN.fbHome.stHmi.nOutputIndex
        p651134158: MAIN.fbHome.fbDOGroupAll.nSize-1
    Scrollbar (43,80 349x30)
        p2245068023: MAIN.fbHome.fbDOGroupAll.nSize-1
        p1057716461: MAIN.fbHome.stHmi.nOutputIndex
    Textfield (533,118 469x28), "%s", text variable: MAIN.fbHome.stHmi.sInput
    Scrollbar (534,79 349x30)
        p2245068023: MAIN.fbHome.fbDIGroupAll.nSize-1
        p1057716461: MAIN.fbHome.stHmi.nInputIndex
    SpinControl (896,80 105x30), variable: MAIN.fbHome.stHmi.nInputIndex
        p651134158: MAIN.fbHome.fbDIGroupAll.nSize-1
    Table (532,154 469x226), data array: MAIN.fbHome.stHmi.aLinkedOutputs
        p3854506369: MAIN.fbHome.stHmi.aLinkedOutputs[INDEX]
        p2232123230: Linked outputs
    Textfield (43,10 955x30), "%d links", text variable: MAIN.fbHome.fbLinkManager.nSize
    Textfield (40,386 470x30), "Check if every output is controlled by one or more inputs"
    Textfield (532,386 470x30), "Check if every input is used at least once"
    Textfield (533,43 468x30), "%d inputs", text variable: MAIN.fbHome.fbDIGroupAll.nSize
    Textfield (43,44 468x30), "%d outputs", text variable: MAIN.fbHome.fbDOGroupAll.nSize
END_VISUALIZATION

// ---- VISUs/Overview.TcVIS
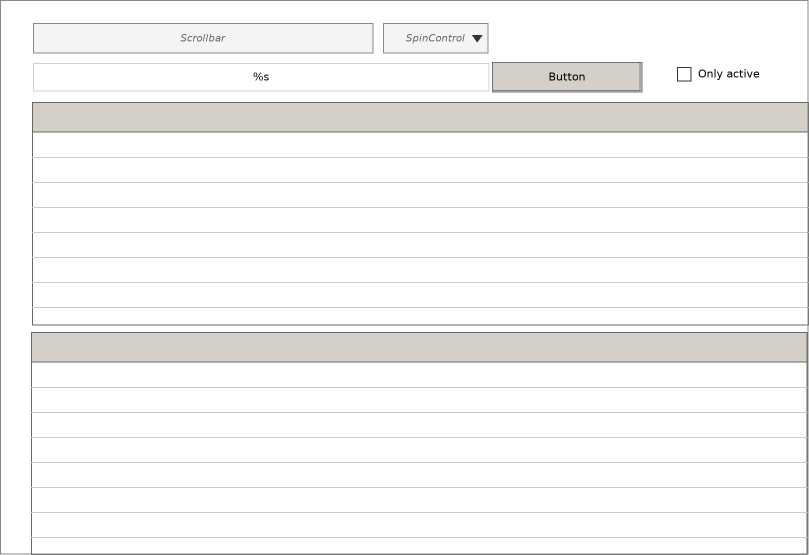
VISUALIZATION Overview  // 809x555
    Button (492,62 150x30), "Button"
        tap MAIN.fbHome.stHmi.bButton
    Table (32,102 777x223), data array: MAIN.fbHome.stHmi.aDigitalIn
        p3854506369: MAIN.fbHome.stHmi.aDigitalIn[INDEX].sName
        p1892666644: MAIN.fbHome.stHmi.aDigitalIn[INDEX].eState
        p338671338: MAIN.fbHome.stHmi.aDigitalIn[INDEX].bValue
    Table (31,332 776x223), data array: MAIN.fbHome.stHmi.aDigitalOut
        p3854506369: MAIN.fbHome.stHmi.aDigitalOut[INDEX].sName
        p1892666644: MAIN.fbHome.stHmi.aDigitalOut[INDEX].eState
        p338671338: MAIN.fbHome.stHmi.aDigitalOut[INDEX].bValue
    SpinControl (383,23 105x30), variable: MAIN.fbHome.stHmi.nInputIndex
        p651134158: MAIN.fbHome.fbDIGroupAll.nSize-1
    Checkbox (675,51 133x46), "Only active", variable: MAIN.fbHome.stHmi.bOnlyActive
    Scrollbar (33,23 340x30)
        p2245068023: MAIN.fbHome.fbDIGroupAll.nSize-1
        p1057716461: MAIN.fbHome.stHmi.nInputIndex
    Textfield (33,63 456x28), "%s", text variable: MAIN.fbHome.stHmi.sInput
END_VISUALIZATION
